{attribute 'linkalways'} 
{attribute 'no_explicit_call' := 'This FB is a CLASS and must be accessed using methods or properties'}
{attribute 'enable_dynamic_creation'}
FUNCTION_BLOCK FINAL Node_NAND EXTENDS Node
VAR
	in1 : _BOOL(FALSE);
    in2 : _BOOL(FALSE);
	out : _BOOL(FALSE);
END_VAR

METHOD PUBLIC  Clone : I_Node
VAR
	pNode : POINTER TO Node_NAND;
END_VAR
pNode := __NEW(Node_NAND);
Clone := pNode^;
END_METHOD

METHOD FB_init : BOOL
VAR_INPUT
	bInitRetains : BOOL; // if TRUE, the retain variables are initialized (warm start / cold start)
	bInCopyCode : BOOL;  // if TRUE, the instance afterwards gets moved into the copy code (online change)
END_VAR
AddParameter('in1', in1);
AddParameter('in2', in2);
AddOutput('out', out);

this^.Metadatum.AddBoolAsMetadata('deprecated', true);
END_METHOD

METHOD PROTECTED OnExecute
VAR
END_VAR
out.Value := NOT(in1.Value AND in2.Value);
END_METHOD

END_FUNCTION_BLOCK

(* stored: Version 1.1.0.1, ProductVersion 3.1.4026.18
   POU Node_NAND: Id {2abc18e9-97dd-0b75-00a0-1883ac5ac979}, SpecialFunc None
   Folder Constructor: Id {c7596e76-6c31-026f-2190-103024a6940b}
   Method Clone: Id {ee3ee99c-f66a-0790-1946-8e5e4ea86c32}
   Method FB_init: Id {3724ad92-9de2-0336-2829-afbacfe17c97}
   Method OnExecute: Id {6e5f3727-bf7b-065a-069d-3813ca4e812a} *)
